// TwinCAT 3 PLC project GitTest
// ProgramVersion: 3.1.4024.12
// libraries:
//   Tc2_Standard, * (Beckhoff Automation GmbH)
//   Tc2_System, * (Beckhoff Automation GmbH)
//   Tc3_Module, * (Beckhoff Automation GmbH)
// project tree:
//   / PlcTask.TcTTO
//   POUs/ FB_Sum.TcPOU, MAIN.TcPOU
// real-time tasks:
//   TASK PlcTask: cycle T#10ms, priority 20, ADS port 350

CONFIGURATION GitTest
    RESOURCE PLC ON TwinCAT3
        TASK PlcTask(INTERVAL := T#10ms, PRIORITY := 20);
        PROGRAM MAIN WITH PlcTask : MAIN;
    END_RESOURCE
END_CONFIGURATION

// ---- POUs/MAIN.TcPOU
PROGRAM MAIN
VAR
	
	a: INT;
	FB_Sum1:FB_Sum;
	num1: INT;
	num2: INT;
	sum1: INT;
END_VAR

a:=a+1;
FB_Sum1(in1:=num1 , in2:=num2 , sum=>sum1 );

END_PROGRAM

// ---- POUs/FB_Sum.TcPOU
FUNCTION_BLOCK FB_Sum
VAR_INPUT
	in1,in2:INT;
END_VAR

VAR_OUTPUT
	sum:INT;
END_VAR
VAR
END_VAR

sum:=in1+in2;

END_FUNCTION_BLOCK
